(* PLC project FromServer, Turbopneumatic Socket Server 1, author DVorobiev *)
(* stored: creationDateTime 2020-11-19T10:39:58, productRelease 1, companyURL www.turbo.ru, modificationDateTime 2020-12-04T14:08:22, version 1, organization Turbopneumatic *)

(* mainServer *)
PROGRAM mainServer
  VAR
    python_eval0 : python_eval;
    trigger : BOOL := False;
    trigger0 : BOOL := False;
    s_out : STRING;
    python_eval1 : python_eval;
  END_VAR

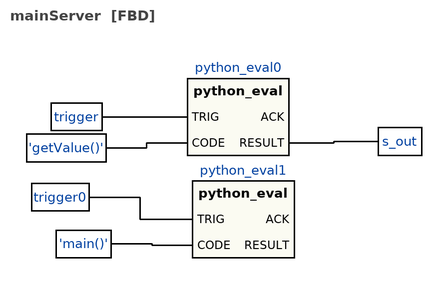
(* FBD diagram, written out as Structured Text *)
python_eval0(TRIG := trigger, CODE := 'getValue()');
s_out := python_eval0.RESULT;
python_eval1(TRIG := trigger0, CODE := 'main()');
END_PROGRAM

CONFIGURATION config
  RESOURCE resource1 ON PLC
    TASK taskServer(INTERVAL := T#1s0ms, PRIORITY := 0);
    PROGRAM srv WITH taskServer : mainServer;
  END_RESOURCE
END_CONFIGURATION
